// TIA Portal V19 export
DATA_BLOCK "PPrgArchive13"   // DB518
// stored: IsOnlyStoredInLoadMemory true, MemoryReserve 0, Namespace G
   VAR RETAIN
      PRG : Array[1201..1300] of "PPrg_Data";
   END_VAR
BEGIN
END_DATA_BLOCK
